{attribute 'pack_mode' := '1'}
    {attribute 'OPC.UA.DA' := '1'}
    {attribute 'OPC.UA.DA.StructuredType' := '1'}
    (*
    ST_RW_InterlockEquipmentMap_HMI_IgnitionExp
    ==================================================
    Generated from Ignition UDT: RW_Interlock_Equipment_Map
    Total tags: 1
    Generated on: 2025-09-15 12:47:18
    *)
    TYPE ST_RW_InterlockEquipmentMap_HMI_IgnitionExp :
    STRUCT
        {attribute 'OPC.UA.DA' := '1'}
        Interlock_Path : STRING := '';
    END_STRUCT
    END_TYPE

(* stored: Version 1.1.0.1
   DUT ST_RW_InterlockEquipmentMap_HMI_IgnitionExp: Id {940f3a32-247e-48a0-aff3-63db75acdd64} *)
